
FUNCTION CB_expt_int : INT


TITLE = ' Exponentiation of a variable  '
VERSION : '1.0'
AUTHOR  : CB
NAME    : exptInt
FAMILY  : TNI

VAR_INPUT
    IN1 : INT;
    IN2 : INT;

END_VAR

BEGIN

CB_expt_int := REAL_TO_INT(IN1 ** IN2);

END_FUNCTION
